PROGRAM MAIN
VAR
	fileToServe : STRING := '/Images/Favicon.ico';
END_VAR

END_PROGRAM

(* stored: Version 1.1.0.1, ProductVersion 3.1.4024.9
   POU MAIN: Id {83e121c2-c55d-4f27-b73a-4e94f5913a2a}, SpecialFunc None *)
